	80:																														// Manual process closing
		Cycle_Stage														:= 'desorption.stopping';
		U.product_vacuum_backfeed_valve									:= _CLOSED;
		rTime1															:= _STOPPING_TIME;
		i7Step															:= 81;
		
	81:
		bTimer1															:= TRUE;
		IF tonTimer1.Q THEN
			bTimer1														:= FALSE;
			i7Step														:= 99;
		END_IF

	90:																														// Automatic process stopping
		Cycle_Stage														:= 'desorption.stopping';
		U.product_vacuum_backfeed_valve									:= _CLOSED;											///@ Close valves & turn off pumps
		rTime1															:= _STOPPING_TIME;
		i7Step															:= 91;
		
	91:
		bTimer1															:= TRUE;
		IF tonTimer1.Q THEN
			bTimer1														:= FALSE;
			i7Step														:= 99;
		END_IF
		
	98:																														// Utility error hold - cleared by P_M01
		i7Step															:= 98;
		
	99:
		IF bStopAfterDesorption THEN
			bStop														:= TRUE;
			Stop_M01_RS													:= TRUE;											// Stop Reactor in P_M01.A_AutoMode
			bStopAfterDesorption										:= FALSE;
		END_IF
		bDesorptionDone													:= TRUE;
		Current_Step													:= 0;
		i7Step															:= 0;
	
END_CASE

IF i7Step > 0 AND i7Step < 80 THEN
	IF bMultiProcess THEN
		IF U.safe_shutdown_error_1 <> '' AND giSafeShutdown1RS = 0 THEN
			sSafeShutdownError1											:= U.safe_shutdown_error_1;
			giSafeShutdown1RS											:= RS_Number;
		ELSIF U.safe_shutdown_error_2 <> '' AND giSafeShutdown23RS = 0 THEN
			sSafeShutdownError2											:= U.safe_shutdown_error_2;
			giSafeShutdown23RS											:= RS_Number;
		ELSIF bDesorptionRSError AND giDesorptionErrorRS = 0 THEN
			bDesorptionRSError											:= FALSE;
			giDesorptionErrorRS											:= RS_Number;
			sMessage													:= gsReactorSetWillStopEvacWillFinishOthersWillCompleteCycle;
		ELSIF (sSafeShutdownError2 <> '' OR sSafeShutdownError3 <> '') AND giSafeShutdown23RS = 0 THEN
			giSafeShutdown23RS											:= RS_Number;
		ELSIF (giDesorptionErrorRS + giSafeShutdown23RS) > 0 THEN
			Stop_Reactor_Set											:= TRUE;
		ELSIF (giEvacuationErrorRS + giSafeShutdown1RS) > 0 THEN
			Cancel_Reactor_Set											:= TRUE;
		ELSIF U.os_air_unsafe_temp THEN																							// 5.e
			bStopAfterDesorption										:= TRUE;
		END_IF
		IF NOT bDesorptionErrorCheck THEN
			IF R_S.steam_header_valve_not_closed THEN
				IF R_S.desorption_high_temp_count > _DESORP_MAX_COUNT THEN														//3.4.3.2_2.b
					bDesorptionErrorCheck								:= TRUE;
					i7Step												:= 25;
				ELSIF R_S.average_reactor_pressure > m01.SP_maximum_safe_reactor_steam_pressure THEN							//3.4.3.2_2.c
					bDesorptionErrorCheck								:= TRUE;
					i7Step												:= 27;
				END_IF
			ELSIF NOT u.product_vacuum_pump_isolation_valve_closed THEN
				IF u.post_condenser_line_temp > u01.SP_maximum_inlet_product_vacuum_temperature THEN							//3.4.3.2_2.d
					bDesorptionErrorCheck								:= TRUE;
					i7Step												:= 28;
				END_IF
			END_IF
		END_IF
	END_IF
	iStep																:= i7Step;
	Current_Step														:= iStep;
	A_Check_Process();
	i7Step																:= iStep;
END_IF
END_ACTION

ACTION A7_Desorption_Auto:
// Phase 0 - FB_Reactor_Set.A7_Desorption_Test
// Rev 1.0 - June 3, 2024

CASE i7Step OF
	
	0:	;
		
	1:
		Cycle_Stage														:= 'desorption.initialize';							
		rTime2															:= m01.SP_steam_pressurization_and_purge_duration * _MINUTES;
		rTime3															:= m01.SP_vacuum_cooling_duration * _MINUTES;
		IF U.utility_error <> '' THEN																						
			sUtilityError												:= U.utility_error;
			sMessage													:= gsSystemCannotRun;
		ELSIF R_S.reactor_pressure_error <> '' THEN
			sReactorError												:= R_S.reactor_pressure_error;
			sMessage													:= gsProcessCannotRun;
		ELSE
			Steam_Service_Req											:= TRUE;
			IF Steam_Service_Assigned THEN 
				U.cooling_line_pre_condenser_valve						:= TRUE;    // XV-01
				U.purge_product_pre_condenser_valve						:= TRUE;	// XV-02
				U.product_vacuum_pump_isolation_valve 					:= TRUE;	// XV-03
				U.product_vacuum_outlet_isolation_valve 				:= TRUE;	// XV-05
				u.product_vacuum_backfeed_valve_mode					:= eManual;
				U.product_vacuum_backfeed_valve							:= 50;		// PCV-01		
				rTime1													:= _VALVE_TIME;
				i7Step													:= i7Step + 1;
			END_IF
		END_IF
			
	2:
		Cycle_Stage														:= 'desorption.prep_purge_lines';
		bTimer1															:= TRUE;	
		bPass1															:= U.cooling_line_pre_condenser_valve_clear;
		bPass2															:= U.purge_product_pre_condenser_valve_clear;
		bPass3															:= U.product_vacuum_pump_isolation_valve_clear;
		bPass4															:= U.product_vacuum_outlet_isolation_valve_clear;
		bPass5															:= NOT  U.product_vacuum_backfeed_valve_closed;
		IF bPass1 AND bPass2 AND bPass3 AND bPass4 AND bPass5 THEN
			bTimer1														:= FALSE;
			rTime1														:= 2 * _MINUTES;				 // need more time ????
			i7Step														:= i7Step + 1;
		ELSIF  tonTimer1.Q THEN
			bTimer1														:= FALSE;
			sUtilityError												:= SEL(bPass1, gsCoolingLinePreCondeserValveError, '');
			sUtilityError												:= SEL(bPass2, gsPurgeProductPreCondenserValverError, sUtilityError);
			sUtilityError												:= SEL(bPass3, gsProductVacuumPumpError, sUtilityError);
			sUtilityError												:= SEL(bPass4, gsProductVacuumOutletIsoValveError, sUtilityError);
			sUtilityError												:= SEL(bPass5, gsProductVacuumBackfeedValveError, sUtilityError);
			sMessage													:= gsSystemWillStop;
		END_IF		
		
	3:
		Cycle_Stage														:= 'desorption.prep_purge_lines';
		bTimer1															:= TRUE;
		IF U.purge_product_line_pres < m01.SP_start_steam_purge_reactor_pressure AND U.pre_condenser_line_pres < m01.SP_start_steam_purge_reactor_pressure THEN
			bTimer1														:= FALSE;
			U.cooling_line_pre_condenser_valve							:= FALSE;	
			rTime1														:= _VALVE_TIME;
			i7Step														:= i7Step + 1;
		ELSIF tonTimer1.Q THEN
			bTimer1														:= FALSE;	
			sUtilityError												:=  'Purge Lines Pressure Not Met ';
			sMessage													:= gsSystemWillStop;
		END_IF
		
	4: 
		Cycle_Stage														:= 'desorption.start_steam_pressurization';	
		bTimer1 														:= TRUE;
		// Verify steam header is at proper temperature and pressure  ???
		bPass1															:= U.boiler_ready;
		bPass2															:= U.boiler_outlet_temp > 100;						//  double check the temp SP !!!!
		bPass3															:= U.cooling_line_pre_condenser_valve_clear;
		IF bPass1 AND bPass2 AND bPass3 THEN
			bTimer1														:= FALSE;
			U.steam_header_volume_total_enable							:= TRUE;
			R_S.steam_control_valve_mode								:= eManual;
			R_S.steam_control_valve										:= _OPEN;				// PCV-01 -> 100%
			R_S.steam_header_valve										:= TRUE;				// XV-07
			i7Step														:= i7Step + 1;
		ELSIF tonTimer1.Q THEN
			bTimer1														:= FALSE;
			sUtilityError												:= SEL(bPass1, 'Steam Header Not at Press ', '');
			sUtilityError												:= SEL(bPass1, 'Steam Header Not at Temp ', sUtilityError);
			sUtilityError												:= SEL(bPass1, gsCoolingLinePreCondeserValveError, sUtilityError);
		END_IF
		
	5: 
		Cycle_Stage														:= 'desorption.steam_pressurization';
		bTimer1 														:= TRUE;
		bTimer2															:= TRUE;													// start timer 2 here ? 
		bPass1															:= 	R_S.steam_header_valve_clear;
		bPass2															:= NOT R_S.steam_control_valve_closed;
		IF bPass1 AND bPass2 THEN
			bTimer1														:= FALSE;			
			i7Step														:= i7Step + 1;
		ELSIF tonTimer1.Q THEN
			bTimer1														:= FALSE;
			sReactorError												:= SEL(bPass1,gsSteamHeaderValveError, '');	
			sReactorError												:= SEL(bPass1,gsSteamControlValveError, sReactorError);	
		END_IF
		
		
	6:
		Cycle_Stage														:= 'desorption.steam_pressurization';
		
		IF R_S.average_reactor_pressure >= m01.SP_maximum_target_steam_pressure THEN
			R_S.purge_valve 											:= TRUE;
			U.product_vacuum_pump_vfd									:= u01.SP_product_vacuum_running_vfd_percent;
			u.product_vacuum_backfeed_valve_mode						:= eManual;
			U.product_vacuum_backfeed_valve								:= u01.SP_product_vacuum_backfeed_valve;
			rTime1														:= _VALVE_TIME;
			i7Step														:= i7Step + 1;
		ELSIF tonTimer2.Q OR R_S.sorbent_high_temp > u01.SP_maximum_reasonable_sorbent_TC_reading THEN 									
			bTimer2 													:= FALSE;
			sReactorError												:= SEL(bPass1,gsSteamFailedToPressurizeReactorError, '');
			sReactorError												:= SEL(bPass1,'Sorbent Temperaure Too High ', '');	
		END_IF
		
	7: 
	
		Cycle_Stage														:= 'desorption.steam_purge';
		bTimer1 														:= TRUE;
		bPass1															:= 	R_S.purge_valve_clear;
		bPass2															:= 	U.product_vacuum_pump_vfd_output> 0;
		bPass3															:=  NOT U.product_vacuum_backfeed_valve_closed;
		
		IF bPass1 AND bPass2 AND bPass3 THEN
			bTimer1														:= FALSE;
			U.drainage_on												:= TRUE;			
			i7Step														:= i7Step + 1;
		ELSIF tonTimer1.Q THEN
			bTimer1														:= FALSE;
			sReactorError												:= SEL(bPass1,gsPurgeValveError, '');	
			sUtilityError												:= SEL(bPass1,gsProductVacuumPumpError,'');	
			sUtilityError												:= SEL(bPass1,gsProductVacuumBackfeedValveError,sUtilityError);	
		END_IF
		
	8:
		Cycle_Stage														:= 'desorption.steam_purge';	
//		bTimer2															:= TRUE;
		IF (U01.SP_mass_flow_totalizer <> 0 AND U01.SP_mass_flow_totalizer >= u01.steam_header_volume_total) OR tonTimer2.Q THEN
			bTimer2														:= FALSE;
			R_S.steam_header_valve											:= FALSE;        // RS - XV01
			R_S.purge_valve													:= FALSE;		 // RS - XV05
			R_S.steam_control_valve_mode									:= eManual;
			R_S.steam_control_valve											:= _CLOSED;		// RS - PCV01
			U.product_vacuum_backfeed_valve_mode							:= eManual;
			U.product_vacuum_backfeed_valve									:= _CLOSED;		// U - PCV01
			U.cooling_line_pre_condenser_valve								:= FALSE;		// U - XV01
			U.purge_product_pre_condenser_valve								:= FALSE;		// U - XV02
			U.product_vacuum_pump_vfd										:= 100;
			U.product_blower_vfd											:= 100;
			R_S.cooling_valve												:= TRUE;
			rTime1														:= _VALVE_TIME;
			i7Step														:= i7Step + 1;
		END_IF
	
	9:
		Cycle_Stage														:= 'desorption.vacuum_cooling_start';	
		bTimer1 														:= TRUE;
		bTimer3															:= TRUE;   
		bPass1 															:= R_S.steam_header_valve_clear;
		bPass2 															:= R_S.purge_valve_clear;
		bPass3															:= NOT R_S.steam_control_valve_closed;
		bPass4 															:= NOT U.product_vacuum_backfeed_valve_closed;
		bPass5															:= U.cooling_line_pre_condenser_valve_clear;
		bPass6															:= U.purge_product_pre_condenser_valve_clear;
		bPass7															:= U.product_vacuum_pump_vfd_output > 0;
		bPass8															:= U.product_blower_vfd_output>0;
		bPass9															:= R_S.cooling_valve_clear;
		IF bPass1 AND bPass2 AND bPass3 AND bPass4 AND bPass5 AND bPass6 AND bPass7 AND bPass8 AND bPass9 THEN
			bTimer1														:= FALSE;			
			i7Step														:= i7Step + 1;
		ELSIF tonTimer1.Q THEN
			bTimer1														:= FALSE;
			sReactorError												:= SEL(bPass1,gsSteamHeaderValveError, '');	
			sReactorError												:= SEL(bPass2,gsPurgeValveError, sReactorError);	
			sReactorError												:= SEL(bPass3,gsSteamControlValveError, sReactorError);
			sUtilityError												:= SEL(bPass4,gsProductVacuumBackfeedValveError,'');	
			sUtilityError												:= SEL(bPass5,gsProductVacuumBackfeedValveError,sUtilityError);	
			sUtilityError												:= SEL(bPass6,gsCoolingLinePreCondeserValveError,sUtilityError);	
			sUtilityError												:= SEL(bPass7,gsPurgeProductPreCondenserValverError,sUtilityError);
			sUtilityError												:= SEL(bPass8,gsProductVacuumPumpError,sUtilityError);
			sUtilityError												:= SEL(bPass9,'Product Blower Error',sUtilityError);
			sReactorError												:= SEL(bPass3,gsCoolingValveError, sReactorError);
		END_IF
		
		
	10:
		IF R_S.sorbent_high_temp <= 58 OR tonTimer3.Q THEN
			R_S.cooling_valve											:= FALSE;
			U.product_vacuum_backfeed_valve								:= 50;
			U.product_vacuum_pump_vfd									:= 50;
			u.product_blower_vfd										:= 0;
			i7Step														:= 99;
		END_IF
		IF U.post_condenser_line_temp > 70 THEN
			sUtilityError												:= SEL(bPass4,gsPostCondenserLineHighTempError,'');
		END_IF
		
	80:																														// Manual process closing
		Cycle_Stage														:= 'desorption.stopping';
		U.product_vacuum_backfeed_valve									:= _CLOSED;
		rTime1															:= _STOPPING_TIME;
		i7Step															:= 81;
		
	81:
		bTimer1															:= TRUE;
		IF tonTimer1.Q THEN
			bTimer1														:= FALSE;
			i7Step														:= 99;
		END_IF

	90:																														// Automatic process stopping
		Cycle_Stage														:= 'desorption.stopping';
		U.product_vacuum_backfeed_valve									:= _CLOSED;											///@ Close valves & turn off pumps
		rTime1															:= _STOPPING_TIME;
		i7Step															:= 91;
		
	91:
		bTimer1															:= TRUE;
		IF tonTimer1.Q THEN
			bTimer1														:= FALSE;
			i7Step														:= 99;
		END_IF
		
	98:																														// Utility error hold - cleared by P_M01
		i7Step															:= 98;
		
	99:
		IF bStopAfterDesorption THEN
			bStop														:= TRUE;
			Stop_M01_RS													:= TRUE;											// Stop Reactor in P_M01.A_AutoMode
			bStopAfterDesorption										:= FALSE;
		END_IF
		bDesorptionDone													:= TRUE;
		IF NOT bMultiProcess THEN
			Steam_Service_Req											:= FALSE;
		END_IF
		U.drainage_on													:= FALSE;
		U.steam_header_volume_total_enable								:= FALSE;
		Current_Step													:= 0;
		i7Step															:= 0;
	
END_CASE

IF i7Step > 0 AND i7Step < 80 THEN
//	IF bMultiProcess THEN
//		IF U.safe_shutdown_error_1 <> '' AND giSafeShutdown1RS = 0 THEN
//			sSafeShutdownError1											:= U.safe_shutdown_error_1;
//			giSafeShutdown1RS											:= RS_Number;
//		ELSIF U.safe_shutdown_error_2 <> '' AND giSafeShutdown23RS = 0 THEN
//			sSafeShutdownError2											:= U.safe_shutdown_error_2;
//			giSafeShutdown23RS											:= RS_Number;
//		ELSIF bDesorptionRSError AND giDesorptionErrorRS = 0 THEN
//			bDesorptionRSError											:= FALSE;
//			giDesorptionErrorRS											:= RS_Number;
//			sMessage													:= gsReactorSetWillStopEvacWillFinishOthersWillCompleteCycle;
//		ELSIF (sSafeShutdownError2 <> '' OR sSafeShutdownError3 <> '') AND giSafeShutdown23RS = 0 THEN
//			giSafeShutdown23RS											:= RS_Number;
//		ELSIF (giDesorptionErrorRS + giSafeShutdown23RS) > 0 THEN
//			Stop_Reactor_Set											:= TRUE;
//		ELSIF (giEvacuationErrorRS + giSafeShutdown1RS) > 0 THEN
//			Cancel_Reactor_Set											:= TRUE;
//		ELSIF U.os_air_unsafe_temp THEN																							// 5.e
//			bStopAfterDesorption										:= TRUE;
//		END_IF
//		IF NOT bDesorptionErrorCheck THEN
//			IF R_S.steam_header_valve_not_closed THEN
//				IF R_S.desorption_high_temp_count > _DESORP_MAX_COUNT THEN														//3.4.3.2_2.b
//					bDesorptionErrorCheck								:= TRUE;
//					i7Step												:= 25;
//				ELSIF R_S.average_reactor_pressure > m01.SP_maximum_safe_reactor_steam_pressure THEN							//3.4.3.2_2.c
//					bDesorptionErrorCheck								:= TRUE;
//					i7Step												:= 27;
//				END_IF
//			ELSIF NOT u.product_vacuum_pump_isolation_valve_closed THEN
//				IF u.post_condenser_line_temp > u01.SP_maximum_inlet_product_vacuum_temperature THEN							//3.4.3.2_2.d
//					bDesorptionErrorCheck								:= TRUE;
//					i7Step												:= 28;
//				END_IF
//			END_IF
//		END_IF
//	END_IF
	iStep																:= i7Step;
	Current_Step														:= iStep;
	A_Check_Process();
	i7Step																:= iStep;
END_IF
END_ACTION

ACTION A7_Desorption_Test_Auto:
// Phase 0 - FB_Reactor_Set.A7_Desorption_Test
// Rev 1.0 - June 3, 2024

CASE i7Step OF
	
	0:	;
		
	1:
		Cycle_Stage														:= 'desorption.initialize';							// 4.a
		rTime1															:= 5 * _SECONDS;
		rTime2															:= m01.SP_steam_pressurization_and_purge_duration * _MINUTES;
		rTime3															:= rTime2 + (m01.SP_vacuum_cooling_duration * _MINUTES);
		Steam_Service_Req												:= TRUE;
		IF Steam_Service_Assigned THEN 
			i7Step															:= i7Step + 1;
		END_IF
		
			
	2:
		bTimer1															:= TRUE;
		IF sita_bits[2].1 THEN 
			bTimer1														:= FALSE;
			i7Step														:= 90;
		ELSIF tonTimer1.Q AND  sita_bits[2].2 THEN 
			bTimer1														:= FALSE;
			sReactorError												:= 'Desorption Error';
			sMessage													:= 'Auto Test';
		END_IF

	
		
	80:																														// Manual process closing
		Cycle_Stage														:= 'desorption.stopping';
		U.product_vacuum_backfeed_valve									:= _CLOSED;
		rTime1															:= _STOPPING_TIME;
		i7Step															:= 81;
		
	81:
		bTimer1															:= TRUE;
		IF tonTimer1.Q THEN
			bTimer1														:= FALSE;
			i7Step														:= 99;
		END_IF

	90:																														// Automatic process stopping
		Cycle_Stage														:= 'desorption.stopping';
		rTime1															:= _STOPPING_TIME;
		i7Step															:= 91;
		
	91:
		bTimer1															:= TRUE;
		IF tonTimer1.Q THEN
			bTimer1														:= FALSE;
			i7Step														:= 99;
		END_IF
		
	98:																														// Utility error hold - cleared by P_M01
		i7Step															:= 98;
		
	99:
		IF bStopAfterDesorption THEN
			bStop														:= TRUE;
			Stop_M01_RS													:= TRUE;											// Stop Reactor in P_M01.A_AutoMode
			bStopAfterDesorption										:= FALSE;
		END_IF
		bDesorptionDone													:= TRUE;
		IF NOT bMultiProcess THEN
			Steam_Service_Req											:= FALSE;
		END_IF
		Current_Step													:= 0;
		i7Step															:= 0;
	
END_CASE

IF i7Step > 0 AND i7Step < 80 THEN
	IF bMultiProcess THEN
		IF U.safe_shutdown_error_1 <> '' AND giSafeShutdown1RS = 0 THEN
			sSafeShutdownError1											:= U.safe_shutdown_error_1;
			giSafeShutdown1RS											:= RS_Number;
		ELSIF U.safe_shutdown_error_2 <> '' AND giSafeShutdown23RS = 0 THEN
			sSafeShutdownError2											:= U.safe_shutdown_error_2;
			giSafeShutdown23RS											:= RS_Number;
		ELSIF bDesorptionRSError AND giDesorptionErrorRS = 0 THEN
			bDesorptionRSError											:= FALSE;
			giDesorptionErrorRS											:= RS_Number;
			sMessage													:= gsReactorSetWillStopEvacWillFinishOthersWillCompleteCycle;
		ELSIF (sSafeShutdownError2 <> '' OR sSafeShutdownError3 <> '') AND giSafeShutdown23RS = 0 THEN
			giSafeShutdown23RS											:= RS_Number;
		ELSIF (giDesorptionErrorRS + giSafeShutdown23RS) > 0 THEN
			Stop_Reactor_Set											:= TRUE;
		ELSIF (giEvacuationErrorRS + giSafeShutdown1RS) > 0 THEN
			Cancel_Reactor_Set											:= TRUE;
		ELSIF U.os_air_unsafe_temp THEN																							// 5.e
			bStopAfterDesorption										:= TRUE;
		END_IF
		IF NOT bDesorptionErrorCheck THEN
			IF R_S.steam_header_valve_not_closed THEN
				IF R_S.desorption_high_temp_count > _DESORP_MAX_COUNT THEN														//3.4.3.2_2.b
					bDesorptionErrorCheck								:= TRUE;
					i7Step												:= 25;
				ELSIF R_S.average_reactor_pressure > m01.SP_maximum_safe_reactor_steam_pressure THEN							//3.4.3.2_2.c
					bDesorptionErrorCheck								:= TRUE;
					i7Step												:= 27;
				END_IF
			ELSIF NOT u.product_vacuum_pump_isolation_valve_closed THEN
				IF u.post_condenser_line_temp > u01.SP_maximum_inlet_product_vacuum_temperature THEN							//3.4.3.2_2.d
					bDesorptionErrorCheck								:= TRUE;
					i7Step												:= 28;
				END_IF
			END_IF
		END_IF
	END_IF
	iStep																:= i7Step;
	Current_Step														:= iStep;
	A_Check_Process();
	i7Step																:= iStep;
END_IF
END_ACTION

END_FUNCTION_BLOCK

(* stored: Version 1.1.0.1, ProductVersion 3.1.4024.12
   POU FB_Reactor_Set: Id {7a14df60-c425-4007-b6c2-e2f870fc0897}, SpecialFunc None
   Action A_Check_Process: Id {6ec7fe9a-742c-414a-a60e-a55eaa5d8982}
   Action A_Clear_Variables: Id {0dbcb2f7-e4a4-40b8-8807-7ed3a1095350}
   Action A_Drain_Reactor_Set: Id {1d4eeb92-89ea-4631-b611-8a78ca35984b}
   Action A_RS_Estop: Id {cf93d1cd-7907-498e-85d2-f3966c7bb4c5}
   Action A_SafeShutdown1: Id {58f17301-1562-48ea-8e64-b48970d6c6b8}
   Action A_SafeShutdown1_Test: Id {22813013-862b-477a-aebe-1f913cf9ad11}
   Action A_SafeShutdown2: Id {0478f4ba-01d4-49ea-b425-2c3385e0af09}
   Action A_SafeShutdown2_Test: Id {364a4e67-4c9d-48d1-b46d-bc8794f2a1ff}
   Action A_SafeShutdown3: Id {90b810eb-e64f-407b-bff1-57ccd17da43f}
   Action A_SafeShutdown3_Test: Id {0f2a7dc4-daa9-42c5-aa00-88efb77213a4}
   Action A1_Idle: Id {f9da58c1-f853-41c1-a061-a5899835c823}
   Action A2_Holding: Id {9e6e43e6-ad7c-4a19-a64f-78b30135e164}
   Action A4_Repressurization: Id {2ecadb33-89a1-48b6-98f5-80de0078733a}
   Action A4_Repressurization_Auto: Id {754a3da5-03af-4044-b9fa-b4481f24ea64}
   Action A4_Repressurization_Test_Auto: Id {d54f4594-5373-4b55-adb1-657d529ab07c}
   Action A5_Adsorption: Id {595711b7-e9f6-47c2-8c76-55c4b171f9d1}
   Action A5_Adsorption_Auto: Id {b320dbf0-895a-4407-bdf8-77442686e4f4}
   Action A5_Adsorption_Test_Auto: Id {7fb8031a-7fe0-460a-9991-2ce1a25466f4}
   Action A6_Evacuation: Id {cd508d62-bd0f-400f-86db-e7e2eaa9a6dc}
   Action A6_Evacuation_Auto: Id {f61283cf-bd53-411a-b295-99a0bade7a7d}
   Action A6_Evacuation_Test_Auto: Id {426572ec-5413-4f00-b5c9-efa47cbb2c8d}
   Action A7_Desorption: Id {5100e4b7-74ae-4062-9ef9-c75826bb55d2}
   Action A7_Desorption_Auto: Id {64b66c6d-be92-49a7-80c1-a34cbffc87f4}
   Action A7_Desorption_Test_Auto: Id {10fe6351-b58a-4f94-86df-2ed2ccdb3398} *)
